TYPE ST_DiagnosticsOptions :
STRUCT
	Enable	: BOOL;
	Period	: TIME;
END_STRUCT
END_TYPE

(* stored: Version 1.1.0.1, ProductVersion 3.1.4024.13
   DUT ST_DiagnosticsOptions: Id {ab43494c-f6dc-02c0-1c85-434d18b585bd} *)
